// TIA Portal V20 export
TYPE "typeCmControlNode"
// stored: Namespace Unit1.Em4
   STRUCT
      interlock : "Unit1.Em4.typeCmControlNodeInterlock";
      command : "Unit1.Em4.typeCmControlNodeCommand";
      softcam : "Unit1.Em4.typeCmControlNodeSoftCam";
   END_STRUCT;
END_TYPE
